{attribute 'qualified_only'}
VAR_GLOBAL
END_VAR

(* stored: Version 1.1.0.1, ProductVersion 3.1.4022.18
   GVL SAFETY_OUT_GLV: Id {4c5076ca-51ca-4e41-8517-776a9cb8cdf5} *)
